TYPE "FCP_IN"
VERSION : 0.1
// Block: FCP_IN
   STRUCT
      EFCStatusWord : EFC_STATUS_WORD;
      EFCExStatusWord : EFC_EX_STATUS_WORD;
      FcPStatusWord : FCP_STATUS_WORD;
      SpeedAct : Word;
      PressureAct : Word;
      CurrentAct : Word;
      ASFWarningCode : Word;
      ASFErrorCode : Word;
   END_STRUCT;

END_TYPE
